(*
    This function blocks aims to pack the EL6688 diagnostic data in MUDPI frames
    and transmit them to Time System using Beckhoffs realtime UDP driver (TF6311). 
    The user of this function blocks needs to do the following in order for the library to work correctly:
    - Initialize the library with configuration parameters
        - Destination IP-address (a multicast address)
        - Destination port
        - Source port
*)

{attribute 'c++_compatible'}
FUNCTION_BLOCK FB_MUDPI_SENDER IMPLEMENTS ITcIoUdpProtocolRecv
VAR_INPUT
		ipAddress : Tc2_System.T_IPv4Addr := '0.0.0.0';
		dest_port : UINT := 10000;
		local_port : UINT := 20000;
		instance_name: STRING := 'undefined';
END_VAR
VAR_OUTPUT
END_VAR
VAR
	(* TF6311 realtime driver parameters *)
    {attribute 'TcInitSymbol'}
    oid : OTCID;
    ipUdp : ITcIoUdpProtocol;
    nReceivedPackets : UINT;
    uLastReceivedIP : T_IP_ADDRESS;
    hrInit : HRESULT;
    hrSend : HRESULT; 
    bSuccessfulInitializationOfRealtimeDriver : BOOL := FALSE; // Indication of whether the realtime driver is properly initialized.
	bEnableSending : BOOL := FALSE; // Indication of whether the sender is active or not.
	
	mudpiPacket : ESO_MUDPI.FB_MudpiPacket(topicId := 300, componentId := 5);
	packet_info : T_PACKET_INFO;
	
	  (* Transmission/communication parameters *)
	_destinationIpAddressString : Tc2_System.T_IPv4Addr;
    _destinationIpAddress : UDINT; // Destination address for the data
    _destinationPort : UINT; // Destination port for the data
    _sourcePort : UINT; // Source port of the data
	
	sLibVersion:	   STRING	:= 'UNKNOWN'; // Library version
	
END_VAR

(*
_destinationIpAddressString := ipAddress;
_destinationPort := dest_port;
_sourcePort := local_port;
*)

IF ipUdp <> 0 THEN
	ipUdp.CheckReceived();
END_IF

UpdateMudpiPacket();

METHOD FB_exit : BOOL
VAR_INPUT
    bInCopyCode : BOOL; // if TRUE, the exit method is called for exiting an instance that is copied afterwards (online change).
END_VAR
IF NOT bInCopyCode THEN // no online change
    IF ipUdp <> 0 THEN
        //ipUdp.UnregisterReceiver(nUdpPort); // Shutdown
        //ipUdp.UnregisterReceiver(nUdpPort); // Shutdown
        FW_SafeRelease(ADR(ipUdp));
        FB_exit := TRUE;
    END_IF
END_IF
END_METHOD

METHOD FB_init : BOOL
VAR_INPUT
    bInitRetains : BOOL; // if TRUE, the retain variables are initialized (warm start / cold start)
    bInCopyCode : BOOL;  // if TRUE, the instance afterwards gets moved into the copy code (online change)
END_VAR

sLibVersion := stLibVersion_ESO_ELT_Utility_Library.sVersion;
_destinationIpAddressString := ipAddress;
_destinationPort := dest_port;
_sourcePort := local_port;

IF NOT bInCopyCode THEN // no online change
	IF ipUdp = 0 AND oid <> 0 THEN
	    hrInit := FW_ObjMgr_GetObjectInstance(	oid:=oid, 
											iid:=TC_GLOBAL_IID_LIST.IID_ITcIoUdpProtocol, 
											pipUnk:=ADR(ipUdp) );
		
		IF SUCCEEDED(hrInit) THEN 
			bSuccessfulInitializationOfRealtimeDriver := TRUE;
		(*
			IF  SUCCEEDED(ipUdp.RegisterReceiver(nUdpPort, THIS^)) THEN //open port
				FB_init := TRUE;
			ELSE 
				FB_init := FALSE; 
				FW_SafeRelease(ADR(ipUdp));
			END_IF
			*)
		END_IF
		
	ELSIF oid = 0 THEN 
		FB_init := FALSE; 
		hrInit := ERR_INVALID_PARAM; 				
	END_IF
END_IF
END_METHOD

METHOD FB_reinit : BOOL
IF (ipUdp <> 0) THEN
    //ipUdp.RegisterReceiver(nUdpPort, THIS^);
    //ipUdp.RegisterReceiver(nUdpPort, THIS^);
    FB_reinit := TRUE;
END_IF
END_METHOD

{attribute 'c++_compatible'}
{attribute 'minimal_input_size' := '4'}
{attribute 'pack_mode' := '4'}
METHOD ReceiveData : HRESULT
VAR_INPUT
	ipAddr	: UDINT;
	udpDestPort	: UINT;
	udpSrcPort	: UINT;
	nData	: UDINT;
	pData	: PVOID;
	pVlan	: POINTER TO ETYPE_VLAN_HEADER := 0;
END_VAR
nReceivedPackets := nReceivedPackets + 1;
uLastReceivedIP.ipAdrInternal := ipAddr;
END_METHOD

(*
    This method carry out the sending of the diagnostic data using the Ethernet network driver.
    The parameters are the array of data to be sent and the timestamp that is required by
	the MUDPI protocol.
*)

METHOD SendData : HRESULT
VAR_INPUT
END_VAR
	 
VAR
	
END_VAR

_DestinationIpAddress := F_IpAddress2Integer(_destinationIpAddressString);
IF ipUdp <> 0 AND bSuccessfulInitializationOfRealtimeDriver = TRUE AND bEnableSending THEN
						   
		// Send Data via UDP
    hrSend := ipUdp.SendData(ipDestAddr := _DestinationIpAddress,
                             udpDestPort := _DestinationPort,
                             udpSrcPort := _SourcePort,
                             nData := mudpiPacket.Size(),
                             pData := mudpiPacket.Data(),
                             bCalcUdpCheckSum := FALSE,
                             pVlan := 0);
    IF SUCCEEDED(hrSend) THEN
        mudpiPacket.IncreaseSampleId();
	END_IF
END_IF


SendData:= hrSend;
END_METHOD

METHOD PUBLIC SetMudpiPayload : BOOL
VAR_INPUT
    payload : POINTER TO BYTE;
    payloadSize : UINT;
END_VAR
SetMudpiPayload := mudpiPacket.SetPayload(payload, payloadSize);
END_METHOD

METHOD PUBLIC SetPacketInfo
VAR_INPUT
    TopicId : UDINT; // MUDPI Topic identity
    ComponentId : UINT; // MUDPI component identity
	Timestamp: LREAL := 0;
END_VAR
packet_info.topicId := TopicId;
packet_info.componentId := ComponentId;
packet_info.timestamp := Timestamp;
UpdateMudpiPacket();
END_METHOD

METHOD PUBLIC SetTimestamp
VAR_INPUT
	Timestamp: LREAL;
END_VAR
packet_info.timestamp := Timestamp;
mudpiPacket.SetTimestamp(packet_info.timestamp);
END_METHOD

{attribute 'c++_compatible'}
{attribute 'minimal_input_size' := '4'}
{attribute 'pack_mode' := '4'}
METHOD TcAddRef : UDINT
END_METHOD

{attribute 'object_name' := 'TcQueryInterface'}
{attribute 'c++_compatible'}
{attribute 'signature_flag' := '33554688'}
{attribute 'pack_mode' := '4'}
{attribute 'show'}
{attribute 'minimal_input_size' := '4'}
METHOD TcQueryInterface : HRESULT
VAR_INPUT
	iid	: REFERENCE TO IID;
	pipItf	: POINTER TO PVOID;
END_VAR
VAR
	ipUdpRecv : ITcIoUdpProtocolRecv;
	ipUnknown : ITcUnknown;	
END_VAR
IF GuidsEqual(ADR(iid), ADR(TC_GLOBAL_IID_LIST.IID_ITcIoUdpProtocolRecv)) THEN
	ipUdpRecv := THIS^; // cast to interface pointer
	pipItf^ := ITCUNKNOWN_TO_PVOID(ipUdpRecv);
	TcAddRef();
	TcQueryInterface := S_OK;
ELSIF GuidsEqual(ADR(iid), ADR(TC_GLOBAL_IID_LIST.IID_ITcUnknown)) THEN
	ipUnknown := THIS^; // cast to interface pointer
	pipItf^ := ITCUNKNOWN_TO_PVOID(ipUnknown);
	TcAddRef();
	TcQueryInterface := S_OK;
ELSE
	TcQueryInterface := E_HRESULTAdsErr.NOINTERFACE ; //Call super if this fb extends some other
END_IF
END_METHOD

{attribute 'c++_compatible'}
{attribute 'minimal_input_size' := '4'}
{attribute 'pack_mode' := '4'}
METHOD TcRelease : UDINT
END_METHOD

METHOD PUBLIC UpdateMudpiPacket
VAR_INPUT
END_VAR

mudpiPacket.SetTopicId(packet_info.topicId);
mudpiPacket.SetComponentId(packet_info.componentId);
mudpiPacket.SetTimestamp(packet_info.timestamp);
END_METHOD

END_FUNCTION_BLOCK

(* stored: Version 1.1.0.1, ProductVersion 3.1.4024.11
   POU FB_MUDPI_SENDER: Id {d4fa8378-d747-4dce-8a97-8096c69a61b2}, SpecialFunc None
   Method FB_exit: Id {256139af-eb6a-40e2-add1-4d29b25826b9}
   Method FB_init: Id {83d25a01-0129-4bef-97b5-4a44ae0095eb}
   Method FB_reinit: Id {1fa3c536-8edb-475b-934d-6290c5c77fc1}
   Method ReceiveData: Id {39a59a53-7085-4ff7-995a-4940f9c5a1ee}
   Method SendData: Id {89a28aaf-565a-42ad-8c47-623bd869c230}
   Method SetMudpiPayload: Id {c7026545-2fea-43a9-9045-5dd6cdcb2d7d}
   Method SetPacketInfo: Id {504b9c4d-df6f-4fef-a0f5-d3628ea4ebed}
   Method SetTimestamp: Id {b7a04a9f-77eb-44e5-947d-afa2e0f3d240}
   Method TcAddRef: Id {35bb0499-a901-46cb-90b9-ee80c5d58f66}
   Method TcQueryInterface: Id {d36fcb78-2ab1-4f3b-8d9e-7deecb5c9b12}
   Method TcRelease: Id {95205f5b-edc6-47e0-aef1-36b47f2eeb1f}
   Method UpdateMudpiPacket: Id {ab579cd6-17d6-48b2-b2c6-bce09a799437} *)
